SUBAPPLICATION Vorsteuerventil_2A (* Subapplication Type *)
  (* Standard: 61499-2 *)
  (* Version 1.0, 2023-01-29, Franz *)
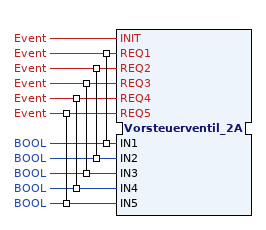
  EVENT_INPUT
    INIT;
    REQ1 WITH IN1;
    REQ2 WITH IN2;
    REQ3 WITH IN3;
    REQ4 WITH IN4;
    REQ5 WITH IN5;
  END_EVENT
  VAR_INPUT
    IN1 : BOOL;
    IN2 : BOOL;
    IN3 : BOOL;
    IN4 : BOOL;
    IN5 : BOOL;
  END_VAR
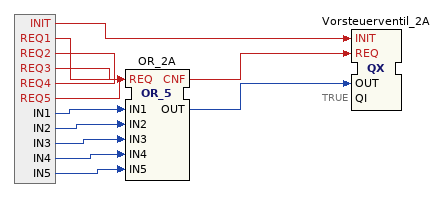
  FBS
    OR_2A : OR_5;
    Vorsteuerventil_2A : QX(QI := TRUE);
  END_FBS
  EVENT_CONNECTIONS
    REQ1 TO OR_2A.REQ;
    REQ2 TO OR_2A.REQ;
    REQ3 TO OR_2A.REQ;
    REQ4 TO OR_2A.REQ;
    REQ5 TO OR_2A.REQ;
    INIT TO Vorsteuerventil_2A.INIT;
    OR_2A.CNF TO Vorsteuerventil_2A.REQ;
  END_CONNECTIONS
  DATA_CONNECTIONS
    IN1 TO OR_2A.IN1;
    IN2 TO OR_2A.IN2;
    IN3 TO OR_2A.IN3;
    IN4 TO OR_2A.IN4;
    IN5 TO OR_2A.IN5;
    OR_2A.OUT TO Vorsteuerventil_2A.OUT;
  END_CONNECTIONS
END_SUBAPPLICATION
